// TIA Portal V17 export
// export: Created 2024-09-02T12:50:20.0190192Z, ExportSetting WithDefaults, DisplayName Totally Integrated Automation Portal, DisplayVersion V17, DisplayName TIA Portal Openness, DisplayVersion V17, DisplayName TIA Portal Version Control Interface, DisplayVersion V17, DisplayName STEP 7 Professional, DisplayVersion V17, DisplayName STEP 7 Safety, DisplayVersion V17, DisplayName WinCC Professional, DisplayVersion V17
FUNCTION "AnwFC2_FG02_Analysis_Status_SLG3_OP70" : Void   // FC1112, LAD
TITLE = Evaluate Moby / Auswerten Moby
{ S7_Optimized_Access := 'TRUE' }
AUTHOR : OlegFuehrus
FAMILY : MOBY
NAME : OlegFuehrus
VERSION : 0.1
// stored: AutoNumber false, IsIECCheckEnabled false, SetENOAutomatically false, UDAEnableTagReadback false
   VAR_TEMP
      t_VKE0 : Bool;   // VKE0
      t_VKE1 : Bool;   // VKE1
      t_Release : Bool;   // Freigabe auswerten / Evaluate release
      t_TafRelease : Array[1..8] of Bool;   // TAF Freigaben / TAF approve
      t_END : Bool;   // Label END
      t_TAFmaske : Byte;
      t_BEA : Array[1..16] of Struct
         General_OK : Bool;
         Prev_OK : Bool;
         Status_OK : Bool;
         Results_OK : Bool;
      END_STRUCT;
      Approve_proces_PreStation : Bool;
      Release_from_MES_BEA : Array[1..8] of Bool;
   END_VAR
   VAR_TEMP   // added for the SCL form of the ladder/FBD networks
      _w1 : Bool;
   END_VAR
BEGIN

REGION Network 1: INIT
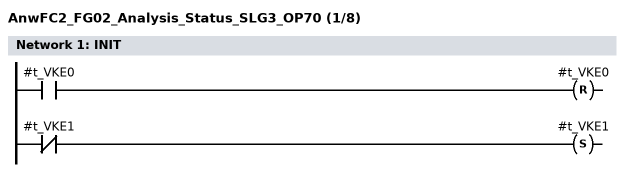
   RUNG wire#powerrail
      Contact( #t_VKE0 )
      R_Coil( #t_VKE0 )
   END_RUNG
   RUNG wire#powerrail
      I_Contact( #t_VKE1 )
      S_Coil( #t_VKE1 )
   END_RUNG
   // the same network as SCL:
   IF #t_VKE0 THEN #t_VKE0 := FALSE; END_IF;
   IF NOT #t_VKE1 THEN #t_VKE1 := TRUE; END_IF;
END_REGION

REGION Network 2: Approve / Reset / Freigabe / Reset
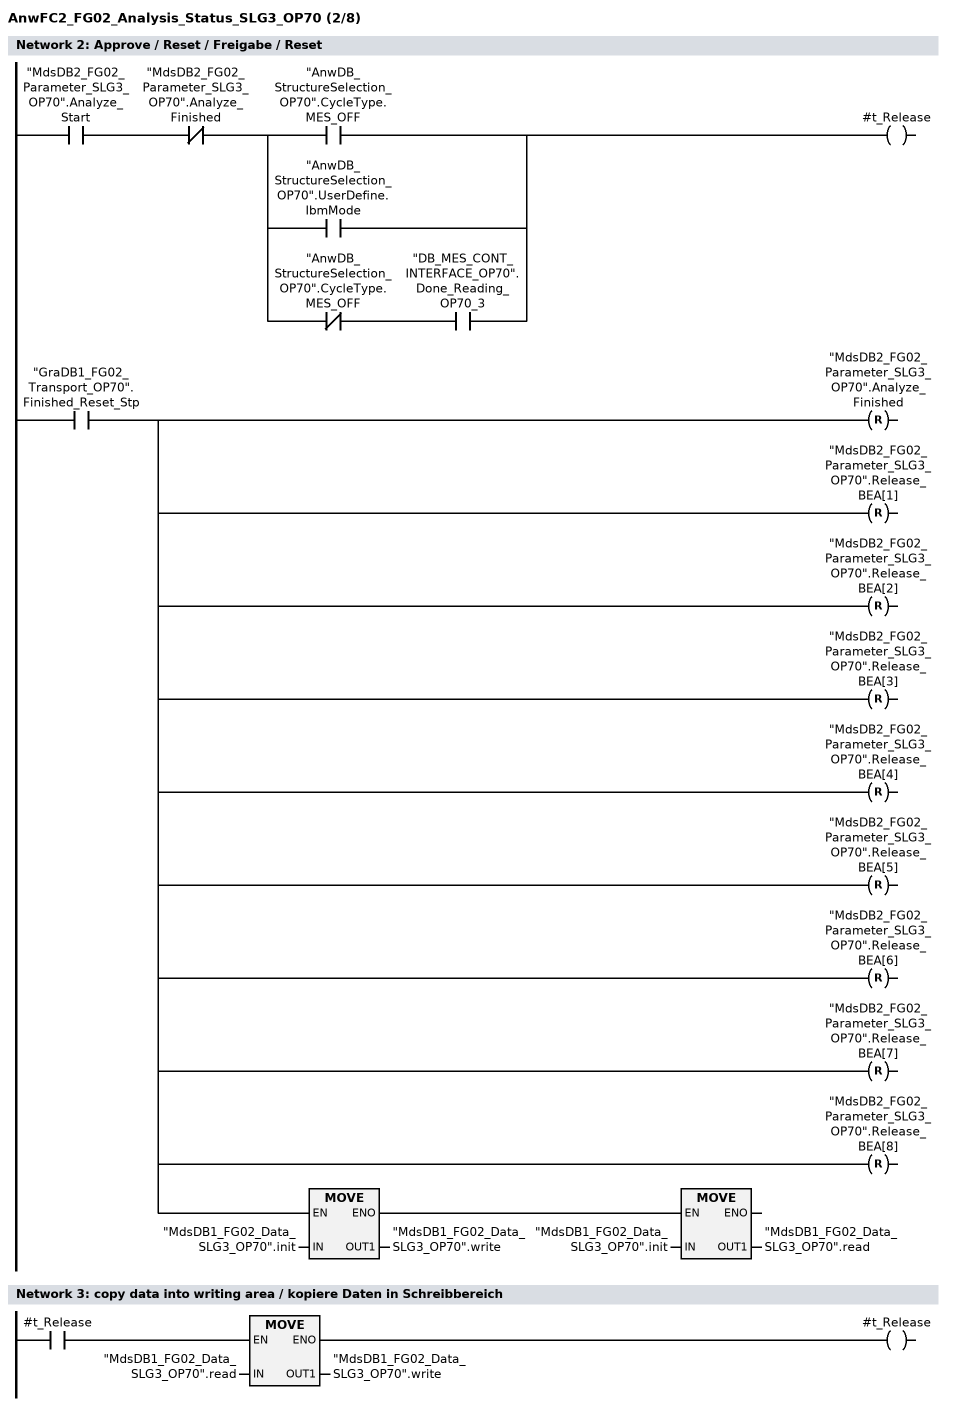
   RUNG wire#powerrail
      Contact( "MdsDB2_FG02_Parameter_SLG3_OP70".Analyze_Start )
      I_Contact( "MdsDB2_FG02_Parameter_SLG3_OP70".Analyze_Finished )
      wire#w1
      Contact( "AnwDB_StructureSelection_OP70".CycleType.MES_OFF )
      wire#w2
      Coil( #t_Release )
   END_RUNG
   RUNG wire#w1
      Contact( "AnwDB_StructureSelection_OP70".UserDefine.IbmMode )
   END_RUNG wire#w2
   RUNG wire#w1
      I_Contact( "AnwDB_StructureSelection_OP70".CycleType.MES_OFF )
      Contact( "DB_MES_CONT_INTERFACE_OP70".Done_Reading_OP70_3 )
   END_RUNG wire#w2
   RUNG wire#powerrail
      Contact( "GraDB1_FG02_Transport_OP70".Finished_Reset_Stp )
      wire#w3
      R_Coil( "MdsDB2_FG02_Parameter_SLG3_OP70".Analyze_Finished )
   END_RUNG
   RUNG wire#w3
      R_Coil( "MdsDB2_FG02_Parameter_SLG3_OP70".Release_BEA[1] )
   END_RUNG
   RUNG wire#w3
      R_Coil( "MdsDB2_FG02_Parameter_SLG3_OP70".Release_BEA[2] )
   END_RUNG
   RUNG wire#w3
      R_Coil( "MdsDB2_FG02_Parameter_SLG3_OP70".Release_BEA[3] )
   END_RUNG
   RUNG wire#w3
      R_Coil( "MdsDB2_FG02_Parameter_SLG3_OP70".Release_BEA[4] )
   END_RUNG
   RUNG wire#w3
      R_Coil( "MdsDB2_FG02_Parameter_SLG3_OP70".Release_BEA[5] )
   END_RUNG
   RUNG wire#w3
      R_Coil( "MdsDB2_FG02_Parameter_SLG3_OP70".Release_BEA[6] )
   END_RUNG
   RUNG wire#w3
      R_Coil( "MdsDB2_FG02_Parameter_SLG3_OP70".Release_BEA[7] )
   END_RUNG
   RUNG wire#w3
      R_Coil( "MdsDB2_FG02_Parameter_SLG3_OP70".Release_BEA[8] )
   END_RUNG
   RUNG wire#w3
      Move(in := "MdsDB1_FG02_Data_SLG3_OP70".init, out1 => "MdsDB1_FG02_Data_SLG3_OP70".write)
      Move(in := "MdsDB1_FG02_Data_SLG3_OP70".init, out1 => "MdsDB1_FG02_Data_SLG3_OP70".read)
   END_RUNG
   // the same network as SCL:
   #t_Release := "MdsDB2_FG02_Parameter_SLG3_OP70".Analyze_Start AND NOT "MdsDB2_FG02_Parameter_SLG3_OP70".Analyze_Finished AND ("AnwDB_StructureSelection_OP70".CycleType.MES_OFF OR "AnwDB_StructureSelection_OP70".UserDefine.IbmMode OR (NOT "AnwDB_StructureSelection_OP70".CycleType.MES_OFF AND "DB_MES_CONT_INTERFACE_OP70".Done_Reading_OP70_3));
   IF "GraDB1_FG02_Transport_OP70".Finished_Reset_Stp THEN
       "MdsDB2_FG02_Parameter_SLG3_OP70".Analyze_Finished := FALSE;
       "MdsDB2_FG02_Parameter_SLG3_OP70".Release_BEA[1] := FALSE;
       "MdsDB2_FG02_Parameter_SLG3_OP70".Release_BEA[2] := FALSE;
       "MdsDB2_FG02_Parameter_SLG3_OP70".Release_BEA[3] := FALSE;
       "MdsDB2_FG02_Parameter_SLG3_OP70".Release_BEA[4] := FALSE;
       "MdsDB2_FG02_Parameter_SLG3_OP70".Release_BEA[5] := FALSE;
       "MdsDB2_FG02_Parameter_SLG3_OP70".Release_BEA[6] := FALSE;
       "MdsDB2_FG02_Parameter_SLG3_OP70".Release_BEA[7] := FALSE;
       "MdsDB2_FG02_Parameter_SLG3_OP70".Release_BEA[8] := FALSE;
       "MdsDB1_FG02_Data_SLG3_OP70".write := "MdsDB1_FG02_Data_SLG3_OP70".init;
       "MdsDB1_FG02_Data_SLG3_OP70".read := "MdsDB1_FG02_Data_SLG3_OP70".init;
   END_IF;
END_REGION

REGION Network 3: copy data into writing area / kopiere Daten in Schreibbereich
   RUNG wire#powerrail
      Contact( #t_Release )
      Move(in := "MdsDB1_FG02_Data_SLG3_OP70".read, out1 => "MdsDB1_FG02_Data_SLG3_OP70".write)
      Coil( #t_Release )
   END_RUNG
   // the same network as SCL:
   IF #t_Release THEN "MdsDB1_FG02_Data_SLG3_OP70".write := "MdsDB1_FG02_Data_SLG3_OP70".read; END_IF;
   #t_Release := #t_Release;
END_REGION

REGION Network 4: Feedback circuit Start / Rückberechnung start
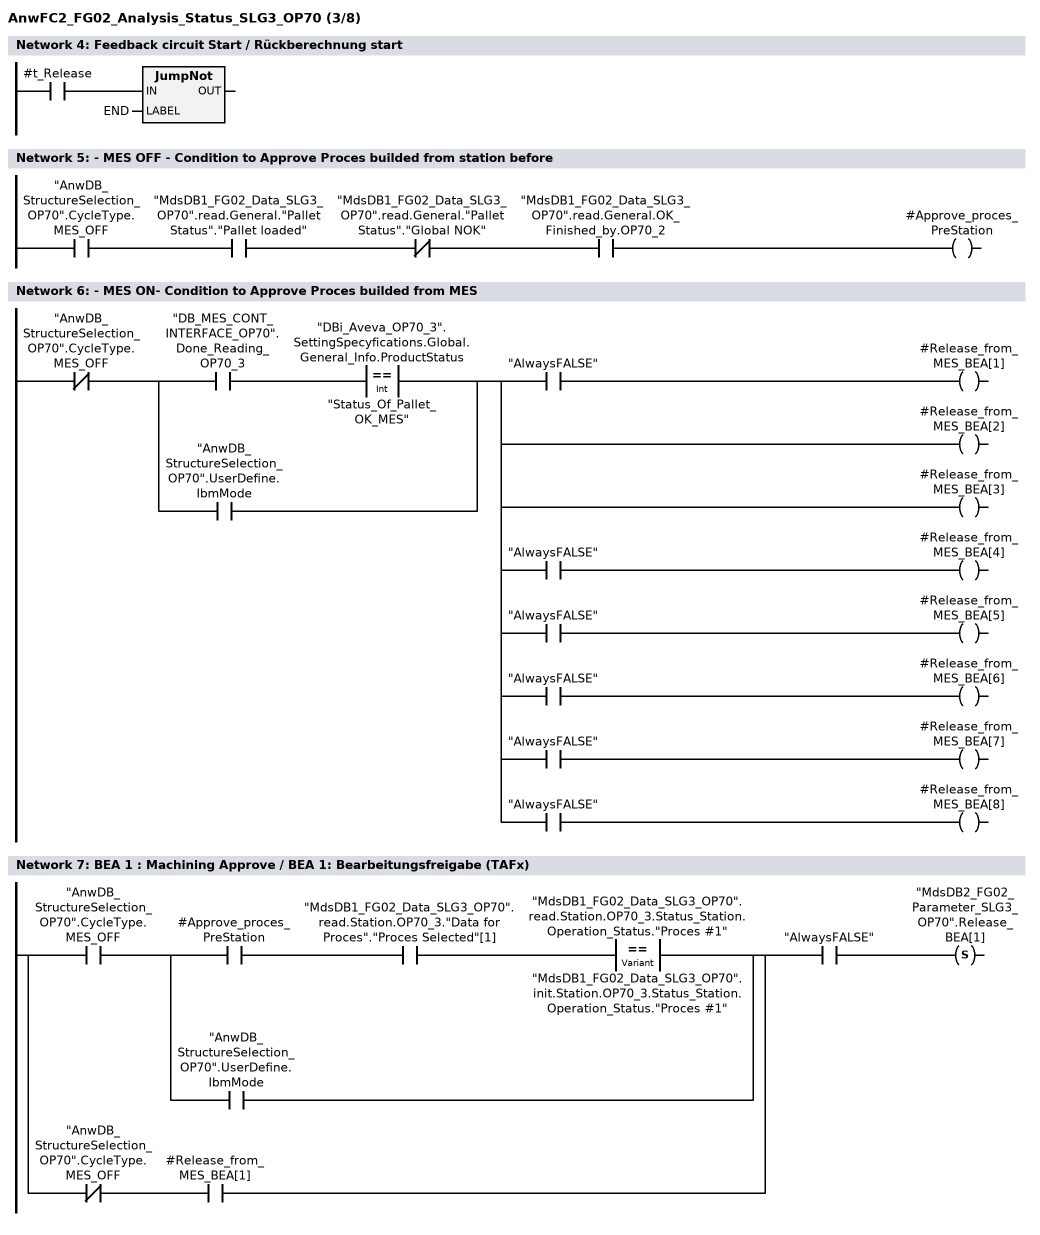
   // no SCL statement known for JumpNot: written as a call
   JumpNot(in := #t_Release, label := END);
END_REGION

REGION Network 5: - MES OFF - Condition to Approve Proces builded from station before
   RUNG wire#powerrail
      Contact( "AnwDB_StructureSelection_OP70".CycleType.MES_OFF )
      Contact( "MdsDB1_FG02_Data_SLG3_OP70".read.General."Pallet Status"."Pallet loaded" )
      I_Contact( "MdsDB1_FG02_Data_SLG3_OP70".read.General."Pallet Status"."Global NOK" )
      Contact( "MdsDB1_FG02_Data_SLG3_OP70".read.General.OK_Finished_by.OP70_2 )
      Coil( #Approve_proces_PreStation )
   END_RUNG
   // the same network as SCL:
   #Approve_proces_PreStation := "AnwDB_StructureSelection_OP70".CycleType.MES_OFF AND "MdsDB1_FG02_Data_SLG3_OP70".read.General."Pallet Status"."Pallet loaded" AND NOT "MdsDB1_FG02_Data_SLG3_OP70".read.General."Pallet Status"."Global NOK" AND "MdsDB1_FG02_Data_SLG3_OP70".read.General.OK_Finished_by.OP70_2;
END_REGION

REGION Network 6: - MES ON- Condition to Approve Proces builded from MES
   RUNG wire#powerrail
      I_Contact( "AnwDB_StructureSelection_OP70".CycleType.MES_OFF )
      wire#w1
      Contact( "DB_MES_CONT_INTERFACE_OP70".Done_Reading_OP70_3 )
      { S7_Templates := "SrcType := Int" } EQ_Contact(in1 := "DBi_Aveva_OP70_3".SettingSpecyfications.Global.General_Info.ProductStatus, in2 := "Status_Of_Pallet_OK_MES")
      wire#w2
      Contact( "AlwaysFALSE" )
      Coil( #Release_from_MES_BEA[1] )
   END_RUNG
   RUNG wire#w1
      Contact( "AnwDB_StructureSelection_OP70".UserDefine.IbmMode )
   END_RUNG wire#w2
   RUNG wire#w2
      Coil( #Release_from_MES_BEA[2] )
   END_RUNG
   RUNG wire#w2
      Coil( #Release_from_MES_BEA[3] )
   END_RUNG
   RUNG wire#w2
      Contact( "AlwaysFALSE" )
      Coil( #Release_from_MES_BEA[4] )
   END_RUNG
   RUNG wire#w2
      Contact( "AlwaysFALSE" )
      Coil( #Release_from_MES_BEA[5] )
   END_RUNG
   RUNG wire#w2
      Contact( "AlwaysFALSE" )
      Coil( #Release_from_MES_BEA[6] )
   END_RUNG
   RUNG wire#w2
      Contact( "AlwaysFALSE" )
      Coil( #Release_from_MES_BEA[7] )
   END_RUNG
   RUNG wire#w2
      Contact( "AlwaysFALSE" )
      Coil( #Release_from_MES_BEA[8] )
   END_RUNG
   // the same network as SCL:
   #_w1 := NOT "AnwDB_StructureSelection_OP70".CycleType.MES_OFF AND (("DB_MES_CONT_INTERFACE_OP70".Done_Reading_OP70_3 AND ("DBi_Aveva_OP70_3".SettingSpecyfications.Global.General_Info.ProductStatus = "Status_Of_Pallet_OK_MES")) OR "AnwDB_StructureSelection_OP70".UserDefine.IbmMode);
   #Release_from_MES_BEA[1] := #_w1 AND "AlwaysFALSE";
   #Release_from_MES_BEA[2] := #_w1;
   #Release_from_MES_BEA[3] := #_w1;
   #Release_from_MES_BEA[4] := #_w1 AND "AlwaysFALSE";
   #Release_from_MES_BEA[5] := #_w1 AND "AlwaysFALSE";
   #Release_from_MES_BEA[6] := #_w1 AND "AlwaysFALSE";
   #Release_from_MES_BEA[7] := #_w1 AND "AlwaysFALSE";
   #Release_from_MES_BEA[8] := #_w1 AND "AlwaysFALSE";
END_REGION

REGION Network 7: BEA 1 : Machining Approve / BEA 1: Bearbeitungsfreigabe (TAFx)
   RUNG wire#powerrail
      Contact( "AnwDB_StructureSelection_OP70".CycleType.MES_OFF )
      wire#w1
      Contact( #Approve_proces_PreStation )
      Contact( "MdsDB1_FG02_Data_SLG3_OP70".read.Station.OP70_3."Data for Proces"."Proces Selected"[1] )
      { S7_Templates := "SrcType := Variant" } EQ_Contact(in1 := "MdsDB1_FG02_Data_SLG3_OP70".read.Station.OP70_3.Status_Station.Operation_Status."Proces #1", in2 := "MdsDB1_FG02_Data_SLG3_OP70".init.Station.OP70_3.Status_Station.Operation_Status."Proces #1")
      wire#w2
      Contact( "AlwaysFALSE" )
      S_Coil( "MdsDB2_FG02_Parameter_SLG3_OP70".Release_BEA[1] )
   END_RUNG
   RUNG wire#w1
      Contact( "AnwDB_StructureSelection_OP70".UserDefine.IbmMode )
   END_RUNG wire#w2
   RUNG wire#powerrail
      I_Contact( "AnwDB_StructureSelection_OP70".CycleType.MES_OFF )
      Contact( #Release_from_MES_BEA[1] )
   END_RUNG wire#w2
   // the same network as SCL:
   IF (("AnwDB_StructureSelection_OP70".CycleType.MES_OFF AND ((#Approve_proces_PreStation AND "MdsDB1_FG02_Data_SLG3_OP70".read.Station.OP70_3."Data for Proces"."Proces Selected"[1] AND ("MdsDB1_FG02_Data_SLG3_OP70".read.Station.OP70_3.Status_Station.Operation_Status."Proces #1" = "MdsDB1_FG02_Data_SLG3_OP70".init.Station.OP70_3.Status_Station.Operation_Status."Proces #1")) OR "AnwDB_StructureSelection_OP70".UserDefine.IbmMode)) OR (NOT "AnwDB_StructureSelection_OP70".CycleType.MES_OFF AND #Release_from_MES_BEA[1])) AND "AlwaysFALSE" THEN
       "MdsDB2_FG02_Parameter_SLG3_OP70".Release_BEA[1] := TRUE;
   END_IF;
END_REGION

REGION Network 8: BEA 2 : Machining Approve / BEA 2: Bearbeitungsfreigabe (TAFx)
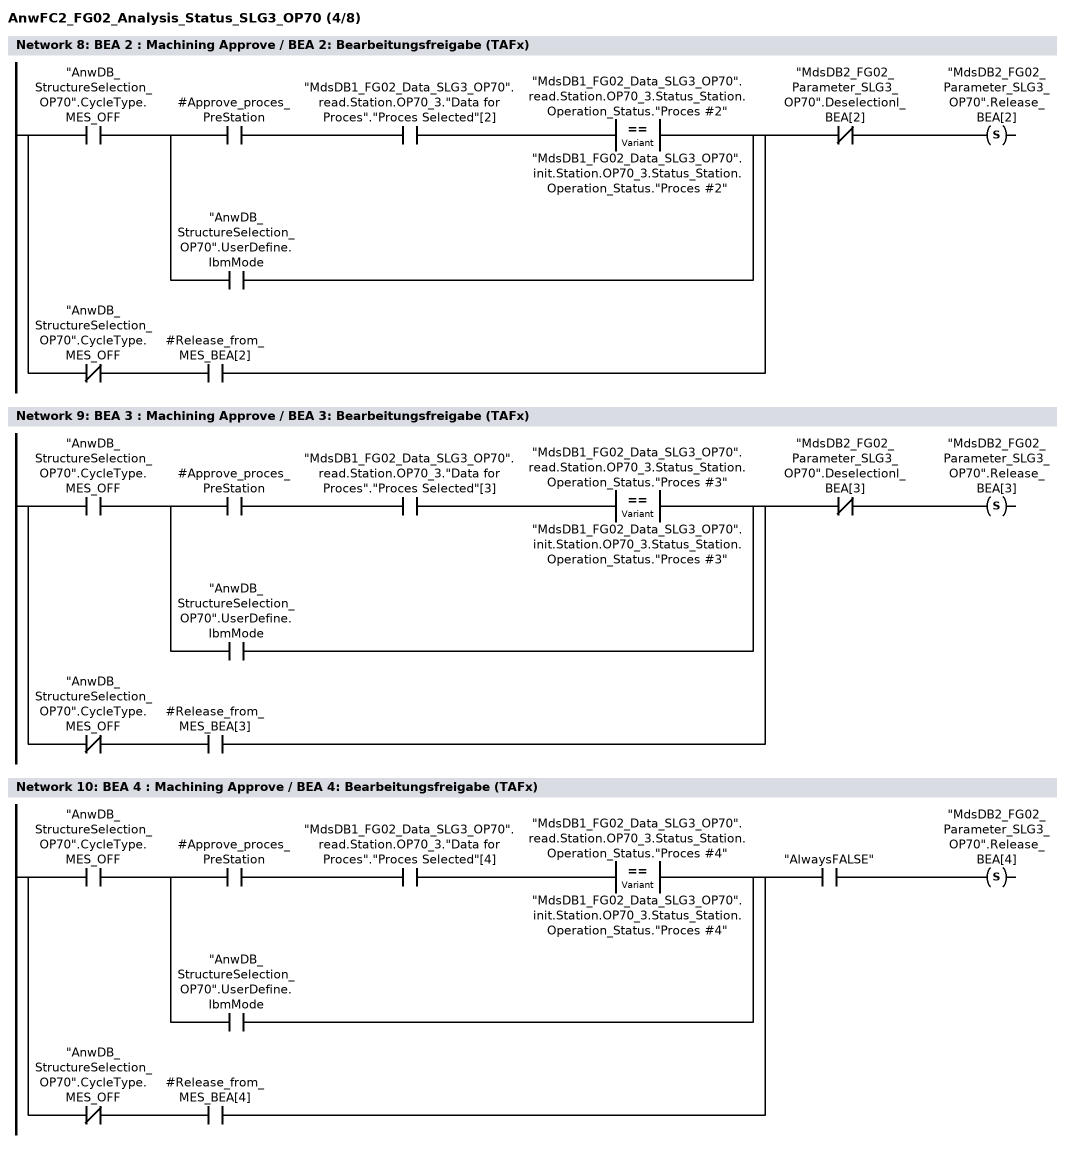
   RUNG wire#powerrail
      Contact( "AnwDB_StructureSelection_OP70".CycleType.MES_OFF )
      wire#w1
      Contact( #Approve_proces_PreStation )
      Contact( "MdsDB1_FG02_Data_SLG3_OP70".read.Station.OP70_3."Data for Proces"."Proces Selected"[2] )
      { S7_Templates := "SrcType := Variant" } EQ_Contact(in1 := "MdsDB1_FG02_Data_SLG3_OP70".read.Station.OP70_3.Status_Station.Operation_Status."Proces #2", in2 := "MdsDB1_FG02_Data_SLG3_OP70".init.Station.OP70_3.Status_Station.Operation_Status."Proces #2")
      wire#w2
      I_Contact( "MdsDB2_FG02_Parameter_SLG3_OP70".Deselectionl_BEA[2] )
      S_Coil( "MdsDB2_FG02_Parameter_SLG3_OP70".Release_BEA[2] )
   END_RUNG
   RUNG wire#w1
      Contact( "AnwDB_StructureSelection_OP70".UserDefine.IbmMode )
   END_RUNG wire#w2
   RUNG wire#powerrail
      I_Contact( "AnwDB_StructureSelection_OP70".CycleType.MES_OFF )
      Contact( #Release_from_MES_BEA[2] )
   END_RUNG wire#w2
   // the same network as SCL:
   IF (("AnwDB_StructureSelection_OP70".CycleType.MES_OFF AND ((#Approve_proces_PreStation AND "MdsDB1_FG02_Data_SLG3_OP70".read.Station.OP70_3."Data for Proces"."Proces Selected"[2] AND ("MdsDB1_FG02_Data_SLG3_OP70".read.Station.OP70_3.Status_Station.Operation_Status."Proces #2" = "MdsDB1_FG02_Data_SLG3_OP70".init.Station.OP70_3.Status_Station.Operation_Status."Proces #2")) OR "AnwDB_StructureSelection_OP70".UserDefine.IbmMode)) OR (NOT "AnwDB_StructureSelection_OP70".CycleType.MES_OFF AND #Release_from_MES_BEA[2])) AND NOT "MdsDB2_FG02_Parameter_SLG3_OP70".Deselectionl_BEA[2] THEN
       "MdsDB2_FG02_Parameter_SLG3_OP70".Release_BEA[2] := TRUE;
   END_IF;
END_REGION

REGION Network 9: BEA 3 : Machining Approve / BEA 3: Bearbeitungsfreigabe (TAFx)
   RUNG wire#powerrail
      Contact( "AnwDB_StructureSelection_OP70".CycleType.MES_OFF )
      wire#w1
      Contact( #Approve_proces_PreStation )
      Contact( "MdsDB1_FG02_Data_SLG3_OP70".read.Station.OP70_3."Data for Proces"."Proces Selected"[3] )
      { S7_Templates := "SrcType := Variant" } EQ_Contact(in1 := "MdsDB1_FG02_Data_SLG3_OP70".read.Station.OP70_3.Status_Station.Operation_Status."Proces #3", in2 := "MdsDB1_FG02_Data_SLG3_OP70".init.Station.OP70_3.Status_Station.Operation_Status."Proces #3")
      wire#w2
      I_Contact( "MdsDB2_FG02_Parameter_SLG3_OP70".Deselectionl_BEA[3] )
      S_Coil( "MdsDB2_FG02_Parameter_SLG3_OP70".Release_BEA[3] )
   END_RUNG
   RUNG wire#w1
      Contact( "AnwDB_StructureSelection_OP70".UserDefine.IbmMode )
   END_RUNG wire#w2
   RUNG wire#powerrail
      I_Contact( "AnwDB_StructureSelection_OP70".CycleType.MES_OFF )
      Contact( #Release_from_MES_BEA[3] )
   END_RUNG wire#w2
   // the same network as SCL:
   IF (("AnwDB_StructureSelection_OP70".CycleType.MES_OFF AND ((#Approve_proces_PreStation AND "MdsDB1_FG02_Data_SLG3_OP70".read.Station.OP70_3."Data for Proces"."Proces Selected"[3] AND ("MdsDB1_FG02_Data_SLG3_OP70".read.Station.OP70_3.Status_Station.Operation_Status."Proces #3" = "MdsDB1_FG02_Data_SLG3_OP70".init.Station.OP70_3.Status_Station.Operation_Status."Proces #3")) OR "AnwDB_StructureSelection_OP70".UserDefine.IbmMode)) OR (NOT "AnwDB_StructureSelection_OP70".CycleType.MES_OFF AND #Release_from_MES_BEA[3])) AND NOT "MdsDB2_FG02_Parameter_SLG3_OP70".Deselectionl_BEA[3] THEN
       "MdsDB2_FG02_Parameter_SLG3_OP70".Release_BEA[3] := TRUE;
   END_IF;
END_REGION

REGION Network 10: BEA 4 : Machining Approve / BEA 4: Bearbeitungsfreigabe (TAFx)
   RUNG wire#powerrail
      Contact( "AnwDB_StructureSelection_OP70".CycleType.MES_OFF )
      wire#w1
      Contact( #Approve_proces_PreStation )
      Contact( "MdsDB1_FG02_Data_SLG3_OP70".read.Station.OP70_3."Data for Proces"."Proces Selected"[4] )
      { S7_Templates := "SrcType := Variant" } EQ_Contact(in1 := "MdsDB1_FG02_Data_SLG3_OP70".read.Station.OP70_3.Status_Station.Operation_Status."Proces #4", in2 := "MdsDB1_FG02_Data_SLG3_OP70".init.Station.OP70_3.Status_Station.Operation_Status."Proces #4")
      wire#w2
      Contact( "AlwaysFALSE" )
      S_Coil( "MdsDB2_FG02_Parameter_SLG3_OP70".Release_BEA[4] )
   END_RUNG
   RUNG wire#w1
      Contact( "AnwDB_StructureSelection_OP70".UserDefine.IbmMode )
   END_RUNG wire#w2
   RUNG wire#powerrail
      I_Contact( "AnwDB_StructureSelection_OP70".CycleType.MES_OFF )
      Contact( #Release_from_MES_BEA[4] )
   END_RUNG wire#w2
   // the same network as SCL:
   IF (("AnwDB_StructureSelection_OP70".CycleType.MES_OFF AND ((#Approve_proces_PreStation AND "MdsDB1_FG02_Data_SLG3_OP70".read.Station.OP70_3."Data for Proces"."Proces Selected"[4] AND ("MdsDB1_FG02_Data_SLG3_OP70".read.Station.OP70_3.Status_Station.Operation_Status."Proces #4" = "MdsDB1_FG02_Data_SLG3_OP70".init.Station.OP70_3.Status_Station.Operation_Status."Proces #4")) OR "AnwDB_StructureSelection_OP70".UserDefine.IbmMode)) OR (NOT "AnwDB_StructureSelection_OP70".CycleType.MES_OFF AND #Release_from_MES_BEA[4])) AND "AlwaysFALSE" THEN
       "MdsDB2_FG02_Parameter_SLG3_OP70".Release_BEA[4] := TRUE;
   END_IF;
END_REGION

REGION Network 11: BEA 5 : Machining Approve / BEA 5: Bearbeitungsfreigabe (TAFx)
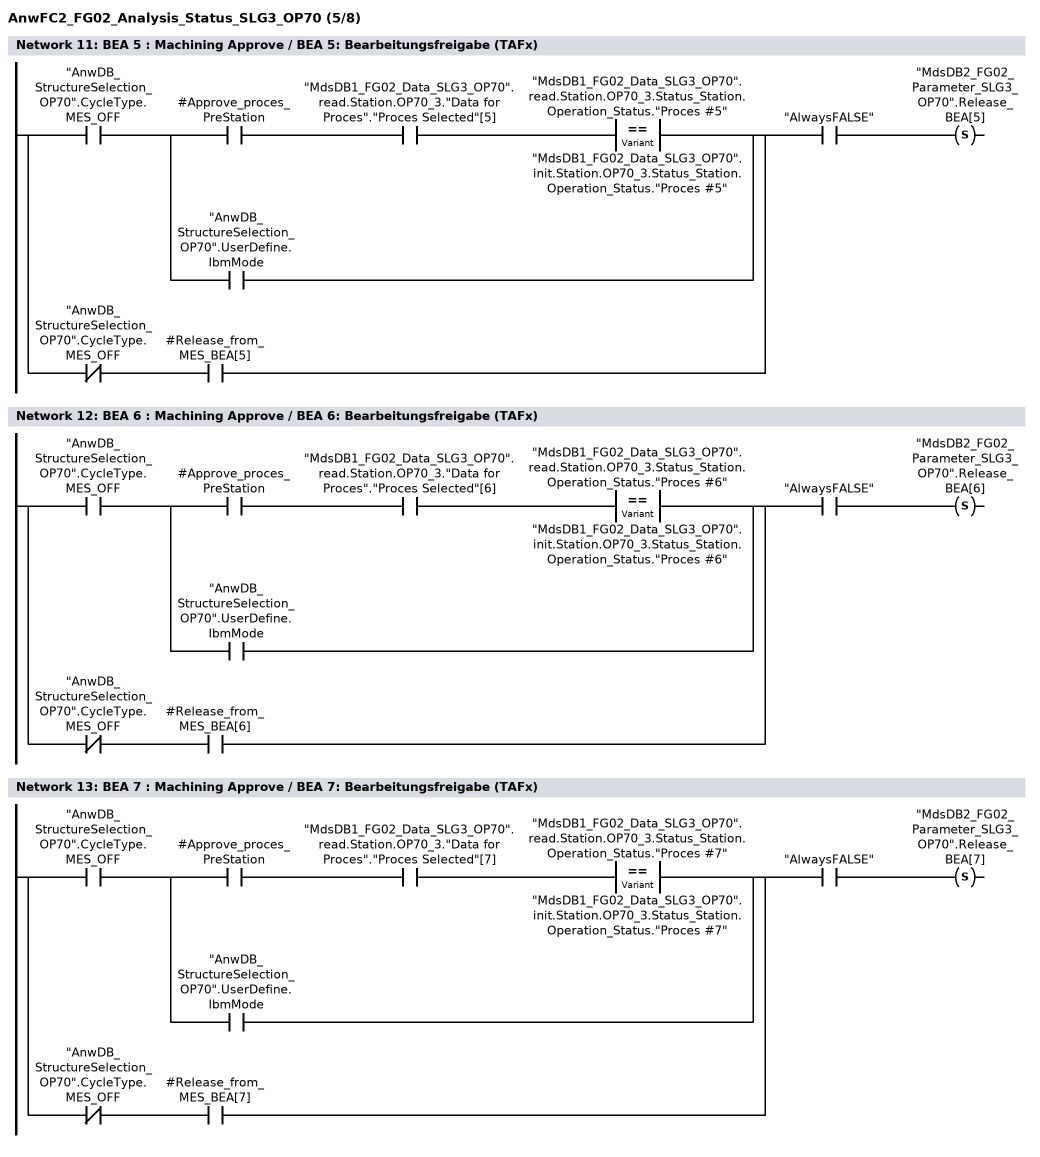
   RUNG wire#powerrail
      Contact( "AnwDB_StructureSelection_OP70".CycleType.MES_OFF )
      wire#w1
      Contact( #Approve_proces_PreStation )
      Contact( "MdsDB1_FG02_Data_SLG3_OP70".read.Station.OP70_3."Data for Proces"."Proces Selected"[5] )
      { S7_Templates := "SrcType := Variant" } EQ_Contact(in1 := "MdsDB1_FG02_Data_SLG3_OP70".read.Station.OP70_3.Status_Station.Operation_Status."Proces #5", in2 := "MdsDB1_FG02_Data_SLG3_OP70".init.Station.OP70_3.Status_Station.Operation_Status."Proces #5")
      wire#w2
      Contact( "AlwaysFALSE" )
      S_Coil( "MdsDB2_FG02_Parameter_SLG3_OP70".Release_BEA[5] )
   END_RUNG
   RUNG wire#w1
      Contact( "AnwDB_StructureSelection_OP70".UserDefine.IbmMode )
   END_RUNG wire#w2
   RUNG wire#powerrail
      I_Contact( "AnwDB_StructureSelection_OP70".CycleType.MES_OFF )
      Contact( #Release_from_MES_BEA[5] )
   END_RUNG wire#w2
   // the same network as SCL:
   IF (("AnwDB_StructureSelection_OP70".CycleType.MES_OFF AND ((#Approve_proces_PreStation AND "MdsDB1_FG02_Data_SLG3_OP70".read.Station.OP70_3."Data for Proces"."Proces Selected"[5] AND ("MdsDB1_FG02_Data_SLG3_OP70".read.Station.OP70_3.Status_Station.Operation_Status."Proces #5" = "MdsDB1_FG02_Data_SLG3_OP70".init.Station.OP70_3.Status_Station.Operation_Status."Proces #5")) OR "AnwDB_StructureSelection_OP70".UserDefine.IbmMode)) OR (NOT "AnwDB_StructureSelection_OP70".CycleType.MES_OFF AND #Release_from_MES_BEA[5])) AND "AlwaysFALSE" THEN
       "MdsDB2_FG02_Parameter_SLG3_OP70".Release_BEA[5] := TRUE;
   END_IF;
END_REGION

REGION Network 12: BEA 6 : Machining Approve / BEA 6: Bearbeitungsfreigabe (TAFx)
   RUNG wire#powerrail
      Contact( "AnwDB_StructureSelection_OP70".CycleType.MES_OFF )
      wire#w1
      Contact( #Approve_proces_PreStation )
      Contact( "MdsDB1_FG02_Data_SLG3_OP70".read.Station.OP70_3."Data for Proces"."Proces Selected"[6] )
      { S7_Templates := "SrcType := Variant" } EQ_Contact(in1 := "MdsDB1_FG02_Data_SLG3_OP70".read.Station.OP70_3.Status_Station.Operation_Status."Proces #6", in2 := "MdsDB1_FG02_Data_SLG3_OP70".init.Station.OP70_3.Status_Station.Operation_Status."Proces #6")
      wire#w2
      Contact( "AlwaysFALSE" )
      S_Coil( "MdsDB2_FG02_Parameter_SLG3_OP70".Release_BEA[6] )
   END_RUNG
   RUNG wire#w1
      Contact( "AnwDB_StructureSelection_OP70".UserDefine.IbmMode )
   END_RUNG wire#w2
   RUNG wire#powerrail
      I_Contact( "AnwDB_StructureSelection_OP70".CycleType.MES_OFF )
      Contact( #Release_from_MES_BEA[6] )
   END_RUNG wire#w2
   // the same network as SCL:
   IF (("AnwDB_StructureSelection_OP70".CycleType.MES_OFF AND ((#Approve_proces_PreStation AND "MdsDB1_FG02_Data_SLG3_OP70".read.Station.OP70_3."Data for Proces"."Proces Selected"[6] AND ("MdsDB1_FG02_Data_SLG3_OP70".read.Station.OP70_3.Status_Station.Operation_Status."Proces #6" = "MdsDB1_FG02_Data_SLG3_OP70".init.Station.OP70_3.Status_Station.Operation_Status."Proces #6")) OR "AnwDB_StructureSelection_OP70".UserDefine.IbmMode)) OR (NOT "AnwDB_StructureSelection_OP70".CycleType.MES_OFF AND #Release_from_MES_BEA[6])) AND "AlwaysFALSE" THEN
       "MdsDB2_FG02_Parameter_SLG3_OP70".Release_BEA[6] := TRUE;
   END_IF;
END_REGION

REGION Network 13: BEA 7 : Machining Approve / BEA 7: Bearbeitungsfreigabe (TAFx)
   RUNG wire#powerrail
      Contact( "AnwDB_StructureSelection_OP70".CycleType.MES_OFF )
      wire#w1
      Contact( #Approve_proces_PreStation )
      Contact( "MdsDB1_FG02_Data_SLG3_OP70".read.Station.OP70_3."Data for Proces"."Proces Selected"[7] )
      { S7_Templates := "SrcType := Variant" } EQ_Contact(in1 := "MdsDB1_FG02_Data_SLG3_OP70".read.Station.OP70_3.Status_Station.Operation_Status."Proces #7", in2 := "MdsDB1_FG02_Data_SLG3_OP70".init.Station.OP70_3.Status_Station.Operation_Status."Proces #7")
      wire#w2
      Contact( "AlwaysFALSE" )
      S_Coil( "MdsDB2_FG02_Parameter_SLG3_OP70".Release_BEA[7] )
   END_RUNG
   RUNG wire#w1
      Contact( "AnwDB_StructureSelection_OP70".UserDefine.IbmMode )
   END_RUNG wire#w2
   RUNG wire#powerrail
      I_Contact( "AnwDB_StructureSelection_OP70".CycleType.MES_OFF )
      Contact( #Release_from_MES_BEA[7] )
   END_RUNG wire#w2
   // the same network as SCL:
   IF (("AnwDB_StructureSelection_OP70".CycleType.MES_OFF AND ((#Approve_proces_PreStation AND "MdsDB1_FG02_Data_SLG3_OP70".read.Station.OP70_3."Data for Proces"."Proces Selected"[7] AND ("MdsDB1_FG02_Data_SLG3_OP70".read.Station.OP70_3.Status_Station.Operation_Status."Proces #7" = "MdsDB1_FG02_Data_SLG3_OP70".init.Station.OP70_3.Status_Station.Operation_Status."Proces #7")) OR "AnwDB_StructureSelection_OP70".UserDefine.IbmMode)) OR (NOT "AnwDB_StructureSelection_OP70".CycleType.MES_OFF AND #Release_from_MES_BEA[7])) AND "AlwaysFALSE" THEN
       "MdsDB2_FG02_Parameter_SLG3_OP70".Release_BEA[7] := TRUE;
   END_IF;
END_REGION

REGION Network 14: BEA 8 : Machining Approve / BEA 8: Bearbeitungsfreigabe (TAFx)
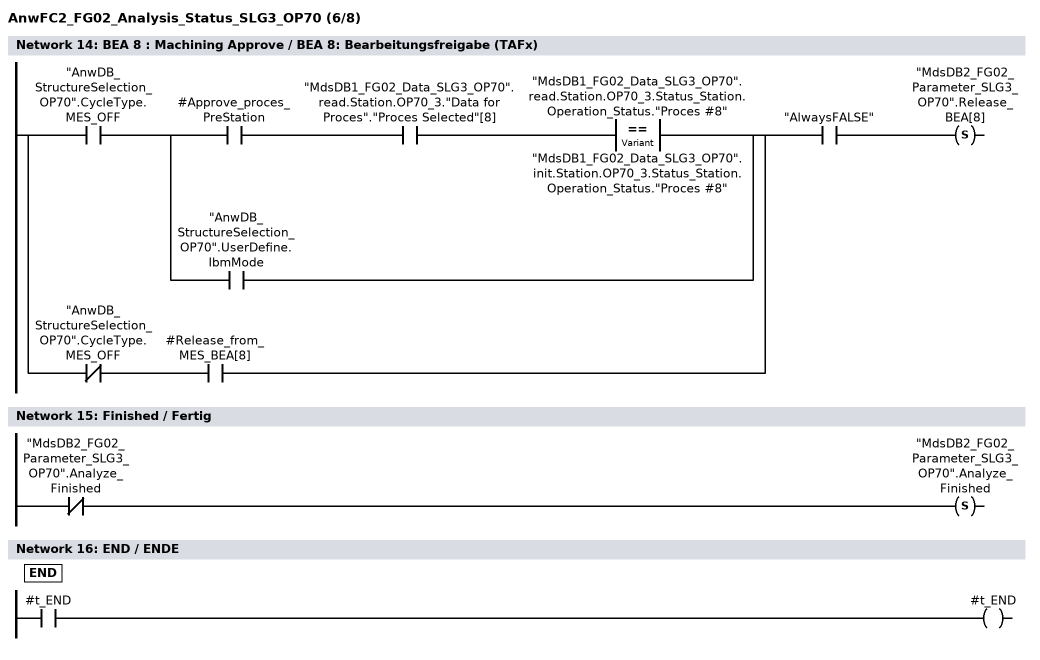
   RUNG wire#powerrail
      Contact( "AnwDB_StructureSelection_OP70".CycleType.MES_OFF )
      wire#w1
      Contact( #Approve_proces_PreStation )
      Contact( "MdsDB1_FG02_Data_SLG3_OP70".read.Station.OP70_3."Data for Proces"."Proces Selected"[8] )
      { S7_Templates := "SrcType := Variant" } EQ_Contact(in1 := "MdsDB1_FG02_Data_SLG3_OP70".read.Station.OP70_3.Status_Station.Operation_Status."Proces #8", in2 := "MdsDB1_FG02_Data_SLG3_OP70".init.Station.OP70_3.Status_Station.Operation_Status."Proces #8")
      wire#w2
      Contact( "AlwaysFALSE" )
      S_Coil( "MdsDB2_FG02_Parameter_SLG3_OP70".Release_BEA[8] )
   END_RUNG
   RUNG wire#w1
      Contact( "AnwDB_StructureSelection_OP70".UserDefine.IbmMode )
   END_RUNG wire#w2
   RUNG wire#powerrail
      I_Contact( "AnwDB_StructureSelection_OP70".CycleType.MES_OFF )
      Contact( #Release_from_MES_BEA[8] )
   END_RUNG wire#w2
   // the same network as SCL:
   IF (("AnwDB_StructureSelection_OP70".CycleType.MES_OFF AND ((#Approve_proces_PreStation AND "MdsDB1_FG02_Data_SLG3_OP70".read.Station.OP70_3."Data for Proces"."Proces Selected"[8] AND ("MdsDB1_FG02_Data_SLG3_OP70".read.Station.OP70_3.Status_Station.Operation_Status."Proces #8" = "MdsDB1_FG02_Data_SLG3_OP70".init.Station.OP70_3.Status_Station.Operation_Status."Proces #8")) OR "AnwDB_StructureSelection_OP70".UserDefine.IbmMode)) OR (NOT "AnwDB_StructureSelection_OP70".CycleType.MES_OFF AND #Release_from_MES_BEA[8])) AND "AlwaysFALSE" THEN
       "MdsDB2_FG02_Parameter_SLG3_OP70".Release_BEA[8] := TRUE;
   END_IF;
END_REGION

REGION Network 15: Finished / Fertig
   RUNG wire#powerrail
      I_Contact( "MdsDB2_FG02_Parameter_SLG3_OP70".Analyze_Finished )
      S_Coil( "MdsDB2_FG02_Parameter_SLG3_OP70".Analyze_Finished )
   END_RUNG
   // the same network as SCL:
   IF NOT "MdsDB2_FG02_Parameter_SLG3_OP70".Analyze_Finished THEN
       "MdsDB2_FG02_Parameter_SLG3_OP70".Analyze_Finished := TRUE;
   END_IF;
END_REGION

REGION Network 16: END / ENDE
   Label( END )
   RUNG wire#powerrail
      Contact( #t_END )
      Coil( #t_END )
   END_RUNG
   // the same network as SCL:
   END:
   #t_END := #t_END;
END_REGION

REGION Network 17: station with -without machining / MOBY: Station mit / ohne Bearbeitung
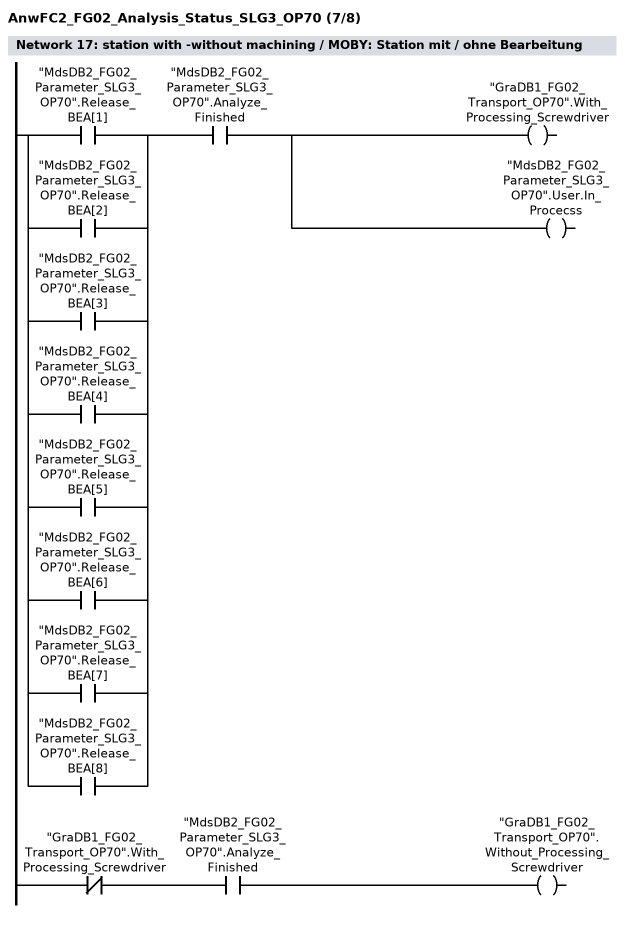
   RUNG wire#powerrail
      Contact( "MdsDB2_FG02_Parameter_SLG3_OP70".Release_BEA[1] )
      wire#w1
      Contact( "MdsDB2_FG02_Parameter_SLG3_OP70".Analyze_Finished )
      wire#w2
      Coil( "GraDB1_FG02_Transport_OP70".With_Processing_Screwdriver )
   END_RUNG
   RUNG wire#powerrail
      Contact( "MdsDB2_FG02_Parameter_SLG3_OP70".Release_BEA[2] )
   END_RUNG wire#w1
   RUNG wire#powerrail
      Contact( "MdsDB2_FG02_Parameter_SLG3_OP70".Release_BEA[3] )
   END_RUNG wire#w1
   RUNG wire#powerrail
      Contact( "MdsDB2_FG02_Parameter_SLG3_OP70".Release_BEA[4] )
   END_RUNG wire#w1
   RUNG wire#powerrail
      Contact( "MdsDB2_FG02_Parameter_SLG3_OP70".Release_BEA[5] )
   END_RUNG wire#w1
   RUNG wire#powerrail
      Contact( "MdsDB2_FG02_Parameter_SLG3_OP70".Release_BEA[6] )
   END_RUNG wire#w1
   RUNG wire#powerrail
      Contact( "MdsDB2_FG02_Parameter_SLG3_OP70".Release_BEA[7] )
   END_RUNG wire#w1
   RUNG wire#powerrail
      Contact( "MdsDB2_FG02_Parameter_SLG3_OP70".Release_BEA[8] )
   END_RUNG wire#w1
   RUNG wire#w2
      Coil( "MdsDB2_FG02_Parameter_SLG3_OP70".User.In_Procecss )
   END_RUNG
   RUNG wire#powerrail
      I_Contact( "GraDB1_FG02_Transport_OP70".With_Processing_Screwdriver )
      Contact( "MdsDB2_FG02_Parameter_SLG3_OP70".Analyze_Finished )
      Coil( "GraDB1_FG02_Transport_OP70".Without_Processing_Screwdriver )
   END_RUNG
   // the same network as SCL:
   "GraDB1_FG02_Transport_OP70".With_Processing_Screwdriver := ("MdsDB2_FG02_Parameter_SLG3_OP70".Release_BEA[1] OR "MdsDB2_FG02_Parameter_SLG3_OP70".Release_BEA[2] OR "MdsDB2_FG02_Parameter_SLG3_OP70".Release_BEA[3] OR "MdsDB2_FG02_Parameter_SLG3_OP70".Release_BEA[4] OR "MdsDB2_FG02_Parameter_SLG3_OP70".Release_BEA[5] OR "MdsDB2_FG02_Parameter_SLG3_OP70".Release_BEA[6] OR "MdsDB2_FG02_Parameter_SLG3_OP70".Release_BEA[7] OR "MdsDB2_FG02_Parameter_SLG3_OP70".Release_BEA[8]) AND "MdsDB2_FG02_Parameter_SLG3_OP70".Analyze_Finished;
   "MdsDB2_FG02_Parameter_SLG3_OP70".User.In_Procecss := "GraDB1_FG02_Transport_OP70".With_Processing_Screwdriver;
   "GraDB1_FG02_Transport_OP70".Without_Processing_Screwdriver := NOT "GraDB1_FG02_Transport_OP70".With_Processing_Screwdriver AND "MdsDB2_FG02_Parameter_SLG3_OP70".Analyze_Finished;
END_REGION

REGION Network 18: Processing enable BEAx / Bearbeitungsfreigabe BEA x
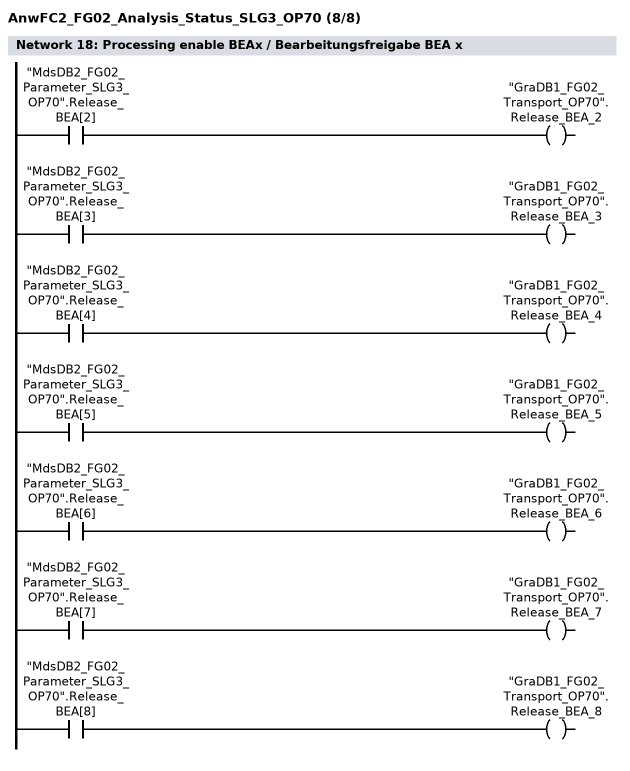
   RUNG wire#powerrail
      Contact( "MdsDB2_FG02_Parameter_SLG3_OP70".Release_BEA[2] )
      Coil( "GraDB1_FG02_Transport_OP70".Release_BEA_2 )
   END_RUNG
   RUNG wire#powerrail
      Contact( "MdsDB2_FG02_Parameter_SLG3_OP70".Release_BEA[3] )
      Coil( "GraDB1_FG02_Transport_OP70".Release_BEA_3 )
   END_RUNG
   RUNG wire#powerrail
      Contact( "MdsDB2_FG02_Parameter_SLG3_OP70".Release_BEA[4] )
      Coil( "GraDB1_FG02_Transport_OP70".Release_BEA_4 )
   END_RUNG
   RUNG wire#powerrail
      Contact( "MdsDB2_FG02_Parameter_SLG3_OP70".Release_BEA[5] )
      Coil( "GraDB1_FG02_Transport_OP70".Release_BEA_5 )
   END_RUNG
   RUNG wire#powerrail
      Contact( "MdsDB2_FG02_Parameter_SLG3_OP70".Release_BEA[6] )
      Coil( "GraDB1_FG02_Transport_OP70".Release_BEA_6 )
   END_RUNG
   RUNG wire#powerrail
      Contact( "MdsDB2_FG02_Parameter_SLG3_OP70".Release_BEA[7] )
      Coil( "GraDB1_FG02_Transport_OP70".Release_BEA_7 )
   END_RUNG
   RUNG wire#powerrail
      Contact( "MdsDB2_FG02_Parameter_SLG3_OP70".Release_BEA[8] )
      Coil( "GraDB1_FG02_Transport_OP70".Release_BEA_8 )
   END_RUNG
   // the same network as SCL:
   "GraDB1_FG02_Transport_OP70".Release_BEA_2 := "MdsDB2_FG02_Parameter_SLG3_OP70".Release_BEA[2];
   "GraDB1_FG02_Transport_OP70".Release_BEA_3 := "MdsDB2_FG02_Parameter_SLG3_OP70".Release_BEA[3];
   "GraDB1_FG02_Transport_OP70".Release_BEA_4 := "MdsDB2_FG02_Parameter_SLG3_OP70".Release_BEA[4];
   "GraDB1_FG02_Transport_OP70".Release_BEA_5 := "MdsDB2_FG02_Parameter_SLG3_OP70".Release_BEA[5];
   "GraDB1_FG02_Transport_OP70".Release_BEA_6 := "MdsDB2_FG02_Parameter_SLG3_OP70".Release_BEA[6];
   "GraDB1_FG02_Transport_OP70".Release_BEA_7 := "MdsDB2_FG02_Parameter_SLG3_OP70".Release_BEA[7];
   "GraDB1_FG02_Transport_OP70".Release_BEA_8 := "MdsDB2_FG02_Parameter_SLG3_OP70".Release_BEA[8];
END_REGION
END_FUNCTION
